// TIA Portal V20 export
TYPE "HMIAxisCtrl_typeInterface"
TITLE = HMIAxisCtrl_typeInterface
// Support: tech.team.motioncontrol@siemens.com 
// Fax: +49 (0) 9131/98-1297
   STRUCT
      actualValues { S7_SetPoint := 'True'} : "HMIAxisCtrl_typeActualValues";   // Actual values of axis
      general { S7_SetPoint := 'True'} : "HMIAxisCtrl_typeGeneral";   // General axis information
      internal { S7_SetPoint := 'True'} : "HMIAxisCtrl_typeInternal";   // Internal variable for visualization
      inputs { S7_SetPoint := 'True'} : "HMIAxisCtrl_typeInputs";   // Inputs AxisCtrl
      outputs { S7_SetPoint := 'True'} : "HMIAxisCtrl_typeOutputs";   // Outputs AxisCtrl
      configuration { S7_SetPoint := 'True'} : "LAxisCtrl_typeAxisConfig";   // Config AxisCtrl
      diagnostics { S7_SetPoint := 'True'} : "LAxisCtrl_typeDiagnostics";   // Diagnostics AxisCtrl
   END_STRUCT;
   // general.axisType := 0;
END_TYPE
